FUNCTION_BLOCK ABSTRACT FB_BaseTelescopeControl IMPLEMENTS I_Telescope
VAR_INPUT
(*
TCS interface section, modeled on an external TCS spec kept as a private internal reference
(not linked here -- this repo is public; ask internally for the spec if you need it). See
specs/design/telescope-telemetry-publish-chain.md for what's actually confirmed about the
on-wire format from tracing the code, since the spec itself isn't accessible from here.
*)
	bPower				: BOOL;		// true: Power on
	bGoHome				: BOOL;		// true: go to home position, unset track/goto if active
	bPark				: BOOL;		// boolean, true: go into park position, ready to stow telescope, unset track/goto
	bTrack				: BOOL;		// boolean, TRUE: MOVE telescope TO last ra/de AND start tracking. Set 'goto' TO FALSE, IF TRUE. FALSE: Stop tracking as soon as possible
	bGoto				: BOOL;		// boolean, TRUE: MOVE telescope TO tau/de AND stop there. Set track TO FALSE, IF TRUE. FALSE: no effect.)	
	bSlew				: BOOL;		// move the telescope to a given az-alt position
	bStop				: BOOL;		// boolean, TRUE: Stop motion OF telescope immediately, set goto AND track TO FALSE. FALSE: Allow motion OF telescope again via track/goto).	
	bReset				: BOOL;		// initiates reset on all axis
	bAutoTrack			: BOOL := TRUE;	// automatic tracking after goto
	bCoverAutoOpen		: BOOL := TRUE;	// automatically open the mirror covers on Init/PowerOn
	// catalog/mean right ascension (ICRS/J2000), degrees, double -- fed straight into AstroBROT's
	// FB_EQ2HOR with precess/nutate/aberration all at their default TRUE, which only makes sense
	// for mean/catalog input (feeding it an already-apparent position would double-correct it);
	// MONETcommon's own telemetry independently re-publishes this same value as *_RA_ICRS (#22)
	fRightAscension		: LREAL :=  0.0;
	// catalog/mean declination (ICRS/J2000), degrees, double -- see fRightAscension
	fDeclination		: LREAL :=  0.0;
	fElevation			: LREAL :=  0.0;	// desired elevation of the telescope pointing
	fAzimuth			: LREAL :=  0.0;	// desired azimut of the telescope pointing
	fTimeOffset			: LREAL := 0.0;		// absolute offset for time
	fHorizon			: LREAL := 1.0;		// ELEVATION below which value the telescope will not go
	
	bEstopTriggered		: BOOL	:= FALSE;	// TODO: CHANGE
	bMainReady			: BOOL	:= TRUE;
	
	telescopeConfig		: ST_TelescopeConfig;
END_VAR
VAR
	fbComm 				: I_Comm;
	
	TCS_command			: E_TCSCommand;	// actual command from the TCS
	fJd					: LREAL;	// current Julian Date calculated from system time
	fLst				: LREAL;	// local siderial time calculated from Julian date in hours
	fElevationCalc		: LREAL;	// elevation calulated when ra and dec are set by TCS 
	fAzimuthCalc		: LREAL;	// azimuth calulated when ra and dec are set by TCS
	fHourAngle			: LREAL;	// hourangle when ra and dec are set by TCS
	
	fRightAscensionCalc	: LREAL;	// right ascension calulated when azimuth and elevation are set by TCS
	fDeclinationCalc	: LREAL;	// declination calulated when azimuth and elevation are set by TCS
	fHourAngleCalc		: LREAL;	// hour angle azimuth and elevation are set by TCS
	
	fbTime				: FB_AstroClock;	// precise astronomical	time
	
	rtrigReset			: R_TRIG;
	bInterrupted		: BOOL;		// If a command is interruped by one with more presedence, the interrupted needs to reset its stage
	
	bPowerFailure		: BOOL;		// triggers power-failure event
	tpPowerOnWarning	: TP;		// triggers power warning
	tonPowerTimeout		: TON;		// power on timeout
	tonCommandTimeout	: TON;		// command timeout
	tonTrackingDelay	: TON;		// tracking delay
	
	TCSpowerEvent,
	TCSgohomeEvent,
	TCSparkEvent,
	TCSgotoEvent,
	TCStrackEvent,
	TCSstopEvent,
	TCStargetHorizonEvent,
	TCSaltitudeEvent,
	TCSnearPoleEvent,
	TCSreadyEvent,
	TCSCTOEvent			: FB_Eventlog;
	tonMQTTTimer 			: TON := (PT:=T#5S);
	// the 7 INFO/CONFIG fields never change at runtime; republishing them on the fast 1-5s
	// telemetry cadence is wasted traffic, so they get their own much slower timer instead
	tonStaticTelemetryTimer	: TON := (PT:=T#30S);
	bStaticTelemetrySent	: BOOL;	// forces one immediate publish on the first cycle
END_VAR
VAR_OUTPUT
	bReady				: BOOL;		// TRUE, IF telescope can be operated 
	fReadyState 		: LREAL := 0.0; // 0: Shut down, 1 powered on, -1 Error
	bIsParked			: BOOL := TRUE;		// telescope is parked
	bIsPowered			: BOOL;		// telescope is powered on
	bError				: BOOL;		// indicates an error on one of the components
	bHorizonError		: BOOL;		// if TRUE, the set Coordinate is below the Horizon threshold fHorizon
	nErrorID				: UDINT;	//error id of axis
	nMotionState		: INT	:= 0;
	bSlewing			: BOOL;		//TRUE, IF telescope is in fast-MOVE phase (includes pole-swap)	
	bTracking			: BOOL;		//TRUE, IF telescope is on tracking position AND currently tracking.	
	bStopped			: BOOL;		//TRUE, IF telescope is AT rest.	
	fHourAngleCurrent	: LREAL;	// true position of the hour angle (without pointing and offset correction)
	fDeclinationCurrent	: LREAL;	// true position of the declination (without pointing and offset correction)
	fRightAscensionCurrent: LREAL;	// true position of the right ascension (without pointing and offset correction)
	fElevationCurrent	: LREAL;	// current position in elevation (calculated) (without pointing and offset correction)
	fAzimuthCurrent		: LREAL;	// current position in azimuth (calculated) (without pointing and offset correction)
	fElevationCurrentSky	: LREAL;	// current position in elevation (calculated)
	fAzimuthCurrentSky		: LREAL;	// current position in azimuth (calculated)
	fSlewTime			: LREAL;	//	(time in sec. to reach the goto/track position) 
	bHomed				: BOOL;		// True: telescope is calibrated
	bBusy				: BOOL;		// telescope does not accept further commands
END_VAR
VAR CONSTANT
	// kept as an inherited constant (not GVL_Math.d2r directly) so existing subclasses
	// (e.g. MONETcommon/MONETN's FB_MonetTelescopeControl) keep working unmodified; single-sourced
	// from GVL_Math now instead of its own copy of PI/180.0
	d2r		: LREAL := GVL_Math.d2r;
END_VAR


// telemetry cadence depends on state: every 1s while slewing/tracking, every 5s otherwise
// (subclasses that don't call SUPER^() from their own cyclic body, e.g. MONETcommon's
// FB_MonetTelescopeControl, drive this on their own timer instead and call _PublishTelemetry()
// directly -- the static-fields gating below lives inside that method, not here, so it still
// applies either way)
IF bSlewing OR bTracking THEN
	tonMQTTTimer.PT := T#1000MS;
ELSE
	tonMQTTTimer.PT := T#5000MS;
END_IF
tonMQTTTimer(IN:=TRUE);
IF tonMQTTTimer.Q THEN
	tonMQTTTimer(IN:=FALSE);
	_PublishTelemetry();
END_IF

METHOD _PublishTelemetry : BOOL
VAR_INPUT
END_VAR
// fbComm is only ever set via FB_Init(comm := ...); nothing enforces that a consumer actually
// does, and calling through an unassigned interface reference crashes the whole PLC task (#7)
IF fbComm = 0 THEN
	RETURN;
END_IF

(* TELESCOPE module*)

//fbComm.Publish('telescope', 'dome', 'TELESCOPE.READY_STATE',	LREAL_TO_STRING(fReadyState));
//fbComm.Publish('telescope', 'dome', 'TELESCOPE.Motion_STATE',	LREAL_TO_STRING(nMotionState));

// static INFO/CONFIG fields never change at runtime: publish once immediately, then only every
// 30s afterward, instead of on every call to this method (#22). Gated here rather than in the
// cyclic body so it still applies when a subclass calls this method directly on its own timer
// instead of going through FB_BaseTelescopeControl's own cyclic body (e.g. MONETcommon's
// FB_MonetTelescopeControl, which never calls SUPER^() from its main body)
tonStaticTelemetryTimer(IN:=TRUE);
IF NOT bStaticTelemetrySent OR tonStaticTelemetryTimer.Q THEN
	tonStaticTelemetryTimer(IN:=FALSE);
	bStaticTelemetrySent := TRUE;
	_PublishStaticTelemetry();
END_IF

// STATUS
IF bEstopTriggered THEN
	fbComm.Publish('telescope', 'dome', 'TELESCOPE.STATUS.GLOBAL', '1');
ELSIF bError THEN
	fbComm.Publish('telescope', 'dome', 'TELESCOPE.STATUS.GLOBAL', '2');
ELSE
	fbComm.Publish('telescope', 'dome', 'TELESCOPE.STATUS.GLOBAL', '0');
END_IF
(* ERROR LIST: TO BE IMPLEMENTED!!!*)

(* OBJECT Module*)

// INSTRUMENTAL
// Set Coords from outside | GoTo:RA DEC | Slew:Alt Az
fbComm.Publish('telescope', 'dome', 'OBJECT.INSTRUMENTAL.RA', LREAL_TO_STRING(fRightAscension));
fbComm.Publish('telescope', 'dome', 'OBJECT.INSTRUMENTAL.DEC', LREAL_TO_STRING(fDeclination));
fbComm.Publish('telescope', 'dome', 'OBJECT.INSTRUMENTAL.ALT', LREAL_TO_STRING(fElevation));
fbComm.Publish('telescope', 'dome', 'OBJECT.INSTRUMENTAL.AZ', LREAL_TO_STRING(fAzimuth));

// HORIZONTAL
IF bSlew THEN
	fbComm.Publish('telescope', 'dome', 'OBJECT.HORIZONTAL.ALT', LREAL_TO_STRING(fElevation));
	fbComm.Publish('telescope', 'dome', 'OBJECT.HORIZONTAL.AZ', LREAL_TO_STRING(fAzimuth));
ELSE
	fbComm.Publish('telescope', 'dome', 'OBJECT.HORIZONTAL.ALT', LREAL_TO_STRING(fElevationCalc));
	fbComm.Publish('telescope', 'dome', 'OBJECT.HORIZONTAL.AZ', LREAL_TO_STRING(fAzimuthCalc));
END_IF

//EQUATORIAL
fbComm.Publish('telescope', 'dome', 'OBJECT.EQUATORIAL.EPOCH', 'J2000.0');
fbComm.Publish('telescope', 'dome', 'OBJECT.EQUATORIAL.EQUINOX', 'J2000.0');
fbComm.Publish('telescope', 'dome', 'OBJECT.EQUATORIAL.RA_PM', '0.0');
fbComm.Publish('telescope', 'dome', 'OBJECT.EQUATORIAL.DEC_PM', '0.0');
fbComm.Publish('telescope', 'dome', 'OBJECT.EQUATORIAL.RA_RATE', '0.0');
fbComm.Publish('telescope', 'dome', 'OBJECT.EQUATORIAL.DEC_RATE', '0.0');
// all angles in the telemetry are degrees, RA included, like the rightascension command (#37)
IF bSlew THEN
	fbComm.Publish('telescope', 'dome', 'OBJECT.EQUATORIAL.RA', LREAL_TO_STRING(fRightAscensionCalc));
	fbComm.Publish('telescope', 'dome', 'OBJECT.EQUATORIAL.DEC', LREAL_TO_STRING(fDeclinationCalc));
ELSE
	fbComm.Publish('telescope', 'dome', 'OBJECT.EQUATORIAL.RA', LREAL_TO_STRING(fRightAscension));
	fbComm.Publish('telescope', 'dome', 'OBJECT.EQUATORIAL.DEC', LREAL_TO_STRING(fDeclination));
END_IF

(*POSITION*)
//LOCAL
fbComm.Publish('telescope', 'dome', 'POSITION.LOCAL.SIDEREAL_TIME', LREAL_TO_STRING(fLst));
fbComm.Publish('telescope', 'dome', 'POSITION.LOCAL.JD', LREAL_TO_STRING(fJd));
fbComm.Publish('telescope', 'dome', 'POSITION.LOCAL.LATITUDE', LREAL_TO_STRING(telescopeConfig.latitude));
fbComm.Publish('telescope', 'dome', 'POSITION.LOCAL.LONGITUDE', LREAL_TO_STRING(telescopeConfig.longitude));
fbComm.Publish('telescope', 'dome', 'POSITION.LOCAL.HEIGHT', LREAL_TO_STRING(telescopeConfig.altitude));
END_METHOD

METHOD _PublishStaticTelemetry : BOOL
VAR_INPUT
END_VAR
// see _PublishTelemetry's identical guard (#7)
IF fbComm = 0 THEN
	RETURN;
END_IF

// fields that never change at runtime -- published on their own slow timer (see the cyclic
// body), not on _PublishTelemetry's fast 1-5s cadence (#22)

// INFO
fbComm.Publish('telescope', 'dome', 'TELESCOPE.INFO.NAME',	telescopeConfig.name);
fbComm.Publish('telescope', 'dome', 'TELESCOPE.INFO.DIAMETER',	LREAL_TO_STRING(telescopeConfig.diameter));
fbComm.Publish('telescope', 'dome', 'TELESCOPE.INFO.CABINET',	telescopeConfig.cabinet);
fbComm.Publish('telescope', 'dome', 'TELESCOPE.INFO.MANUFACTURER', telescopeConfig.manufacturer);

// CONFIG
fbComm.Publish('telescope', 'dome', 'TELESCOPE.CONFIG.CAPABILITIES', '0'); // no ST_TelescopeConfig field for this yet
fbComm.Publish('telescope', 'dome', 'TELESCOPE.CONFIG.MOUNTOPTIONS', telescopeConfig.mountOptions);
fbComm.Publish('telescope', 'dome', 'TELESCOPE.CONFIG.MOUNT', telescopeConfig.mount);
END_METHOD

PROPERTY Altitude : LREAL
GET
Altitude := THIS^.fElevationCurrent;
END_GET
END_PROPERTY

PROPERTY Azimuth : LREAL
GET
Azimuth := THIS^.fAzimuthCurrent;
END_GET
END_PROPERTY

PROPERTY CoverAutoOpen : BOOL
GET
CoverAutoOpen := THIS^.bCoverAutoOpen;
END_GET
SET
THIS^.bCoverAutoOpen := CoverAutoOpen;
END_SET
END_PROPERTY

PROPERTY Declination : LREAL
GET
Declination := THIS^.fDeclinationCurrent;
END_GET
END_PROPERTY

METHOD FB_init : BOOL
VAR_INPUT
	bInitRetains : BOOL; // if TRUE, the retain variables are initialized (warm start / cold start)
	bInCopyCode : BOOL;  // if TRUE, the instance afterwards gets moved into the copy code (online change)
	comm			: I_Comm;	
END_VAR
THIS^.fbComm := comm;
END_METHOD

METHOD Home : BOOL
bGoHome := TRUE;
END_METHOD

METHOD Init : BOOL
bPower := TRUE;
END_METHOD

METHOD Park : BOOL
bPark := TRUE;
END_METHOD

METHOD Reset : BOOL
VAR_INPUT
END_VAR
bReset := TRUE;
END_METHOD

PROPERTY RightAscension : LREAL
GET
RightAscension := THIS^.fRightAscensionCurrent;
END_GET
END_PROPERTY

METHOD Slew : BOOL
VAR_INPUT
	fAzimuth		: LREAL;
	fAltitude		: LREAL;
END_VAR
THIS^.fAzimuth := fAzimuth;
THIS^.fElevation := fAltitude;
bSlew := TRUE;
END_METHOD

METHOD Stop : BOOL
bStop := TRUE;
END_METHOD

METHOD Track : BOOL
VAR_INPUT
	fRightAscension	: LREAL;
	fDeclination	: LREAL;
END_VAR
THIS^.fRightAscension := fRightAscension;
THIS^.fDeclination := fDeclination;
bTrack := TRUE;
END_METHOD

END_FUNCTION_BLOCK

(* stored: Version 1.1.0.1, ProductVersion 3.1.4024.15
   POU FB_BaseTelescopeControl: Id {eddbf876-a986-4fe1-ba5b-16d782882b92}, SpecialFunc None
   Method _PublishTelemetry: Id {6dec3368-4b87-4c9c-96fd-ac4ed46b70ff}
   Method _PublishStaticTelemetry: Id {9c1b6e2a-7f34-4d8e-a5b1-3e6f8c2d9a47}
   Property Altitude: Id {caafb587-dfec-4075-98b5-4e0c659dd422}
   Get Get: Id {3eadfa0f-91b9-4d35-b2a2-3995bf1ad272}
   Property Azimuth: Id {4ab08aee-62ef-436f-afb0-a92312153ecc}
   Get Get: Id {5db7deaa-4ebd-480d-94f2-987ee6c7533c}
   Property CoverAutoOpen: Id {3c28b3ed-e389-4aa6-bf2e-ea34582ac892}
   Get Get: Id {890ef1c5-180f-4a4d-82f6-339804b8a614}
   Set Set: Id {ba214e39-5a4f-40c3-9e98-38c9bb231473}
   Property Declination: Id {f1005b84-337c-4b64-b7ea-204360ce618d}
   Get Get: Id {f2fb9d57-e433-4c82-b5be-80f2fdab955e}
   Method FB_init: Id {a32d2f32-4a31-4d05-8712-e937ed61ba13}
   Method Home: Id {84524932-267e-412f-a6c3-40e991630e8d}
   Method Init: Id {3aef494f-7f4e-4344-8ab1-5311c283fa00}
   Method Park: Id {621c0fc8-dd4d-44e7-85fe-cb7551b9d3ae}
   Method Reset: Id {3d17fa40-fd53-4e7d-b2aa-5ea6dd1055c0}
   Property RightAscension: Id {479a6a93-35a2-4327-9015-03d6802f2b56}
   Get Get: Id {cd895a36-325d-498a-95c9-5d78816a7d56}
   Method Slew: Id {c9fecd44-6a6f-4a55-81c4-7243946a8163}
   Method Stop: Id {8e159726-2715-4778-83ca-31c01953b46c}
   Method Track: Id {edf3f645-ab28-47ec-8a4c-398c458de728} *)
